// Alias for INT values.
// | Result >= 1 - Ok/Success
// | Result = 0 - None
// | Result <=- 1 - Error
TYPE Result : INT; END_TYPE

(* stored: Version 1.1.0.1
   DUT Result: Id {9ee79853-7af1-43d3-abf3-b0e74ce1279f} *)
